TYPE ST_WaferTransferStatus :
STRUCT
	// Process Station identity; zero means no Station is selected for this direction.
	StationId : UDINT;
	Status : ST_ServiceStatus;
	Signal : ST_TransferHandshakeSignal;
END_STRUCT
END_TYPE

(* stored: Version 1.1.0.1, ProductVersion 3.1.4026.18
   DUT ST_WaferTransferStatus: Id {5445009c-02f9-4817-8fcd-e0f304207b54} *)
